PROGRAM MAIN
VAR
	Power: BOOL;
	Initalisatie_voltooid: BOOL;
	Initaliseren: BOOL;
	Tekst: WSTRING(INT#22) := "Hoi" ;
END_VAR

IF Power := TRUE THEN Tekst:= "Initaliseer de machine";
	
END_IF

END_PROGRAM

(* stored: Version 1.1.0.1, ProductVersion 3.1.4024.12
   POU MAIN: Id {4c18c0eb-3271-4093-a9fa-bc44a8c4f230}, SpecialFunc None *)
